{attribute 'no_explicit_call' := 'do not call this POU directly'} 
FUNCTION_BLOCK DigitalOutput_NO
VAR
	output					AT %Q*: BOOL;
END_VAR

METHOD Off : BOOL
output					:= FALSE;
END_METHOD

METHOD On : BOOL
output					:= TRUE;
END_METHOD

PROPERTY status : bool
GET
status				:= output;
END_GET
END_PROPERTY

END_FUNCTION_BLOCK

(* stored: Version 1.1.0.1
   POU DigitalOutput_NO: Id {6f3867cc-4101-47b8-bd6a-182185a54740}, SpecialFunc None
   Method Off: Id {aa084217-960c-48f3-927b-c052c043ac2c}
   Method On: Id {4c61640f-6ff4-4dcc-a976-5e0b12c99cf5}
   Property status: Id {25d672f7-b376-4b0a-a782-1c94882d9b65}
   Get Get: Id {c320242a-9b19-4bb6-8e78-6c3bc17e0747} *)
